TYPE Handshake_Send :
STRUCT
	WaitingToSend	: BOOL;
	Sending			: BOOL;
	PartInfo		: STRING(20);
END_STRUCT
END_TYPE

(* stored: Version 1.1.0.1, ProductVersion 3.1.4022.11
   DUT Handshake_Send: Id {f9b656a8-9dc5-41b8-829d-96bb34d32b5f} *)
